{attribute 'qualified_only'}
{attribute 'strict'}
{attribute 'to_string'}
TYPE E_ConveyorState :
(
	IDLE,
    RUNNING,
    RUNNING_OUT,
    LOCKOUT
);
END_TYPE

(* stored: Version 1.1.0.1
   DUT E_ConveyorState: Id {cccca535-f2fd-4198-a0b6-8fe622c93fb7} *)
